TYPE sss : DATE_AND_TIME
;
END_TYPE

(* stored: Version 1.1.0.1, ProductVersion 3.1.4024.16
   DUT sss: Id {69bf82aa-533a-45c6-b8fb-dec09511ed3d} *)
